PROGRAM A03_StartupLogger
VAR
	fbStartLogger: NT_StartProcess;
	fbPulse: FB_SquareWave;
	tonNotRunning: TON;
	bBusyOnce	:BOOL;

	ton_Watchdog: TON;
	nLastWatchdogFromLogger	: DINT;
	bWait: BOOL;

	bLoggerLocalRun : BOOL;

END_VAR

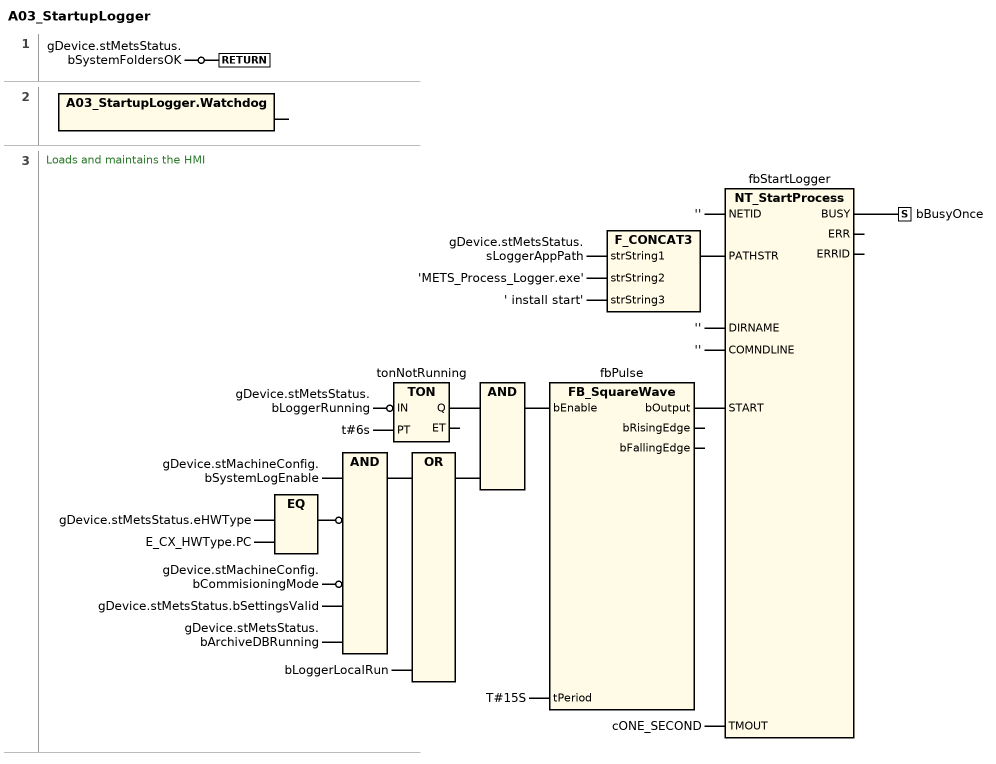
// NETWORK 1
IF NOT gDevice.stMetsStatus.bSystemFoldersOK THEN RETURN; END_IF

// NETWORK 2
A03_StartupLogger.Watchdog();

// NETWORK 3
// Loads and maintains the HMI
tonNotRunning(IN := NOT gDevice.stMetsStatus.bLoggerRunning, PT := t#6s); // TON
fbPulse(bEnable := tonNotRunning.Q AND (gDevice.stMachineConfig.bSystemLogEnable AND NOT (gDevice.stMetsStatus.eHWType = E_CX_HWType.PC) AND NOT gDevice.stMachineConfig.bCommisioningMode AND gDevice.stMetsStatus.bSettingsValid AND gDevice.stMetsStatus.bArchiveDBRunning OR bLoggerLocalRun), tPeriod := T#15S); // FB_SquareWave
fbStartLogger(
    NETID := '',
    PATHSTR := F_CONCAT3(strString1 := gDevice.stMetsStatus.sLoggerAppPath, strString2 := 'METS_Process_Logger.exe', strString3 := ' install start'),
    DIRNAME := '',
    COMNDLINE := '',
    START := fbPulse.bOutput,
    TMOUT := cONE_SECOND); // NT_StartProcess
bBusyOnce S= fbStartLogger.BUSY;

ACTION Watchdog:
(*Watchdog to Bridge*)
gDevice.nWatchdogToLogger := gDevice.nWatchdogToLogger + 1;
IF  gDevice.nWatchdogToLogger > 10000 THEN
	gDevice.nWatchdogToLogger := 1;
END_IF

gDevice.nWatchdogFromLogger	:=	gDevice.stProcessLogger.nLoggerWatchdog;
(*Watchdog from HMI - check if running*)
IF ton_Watchdog.Q THEN
	bWait := FALSE;
	IF gDevice.nWatchdogFromLogger <> nLastWatchdogFromLogger THEN
		gDevice.stMetsStatus.bLoggerRunning := TRUE;
		nLastWatchdogFromLogger := gDevice.nWatchdogFromLogger;
	ELSE
		gDevice.stMetsStatus.bLoggerRunning := FALSE;
	END_IF
ELSE
	bWait := TRUE;
END_IF

ton_Watchdog(IN:= bWait, PT := t#4000ms);
END_ACTION

END_PROGRAM

(* stored: Version 1.1.0.1
   POU A03_StartupLogger: Id {2290d6e2-000e-447f-94b5-cd1b2d7704b7}, SpecialFunc None
   Action Watchdog: Id {5a4c67d7-eef6-4bbe-aa25-aedc885f3c80} *)
